TYPE CHAR : STRING(1); END_TYPE

(* stored: Version 1.1.0.1, ProductVersion 3.1.4024.11
   DUT CHAR: Id {82ab8390-a38a-4ea1-8dc7-eafc65c58e7e} *)
